(* IEC 61131-3 sources: Lasal/CPU_5344_V01/Class/Uitv_Regel_C, 1 file *)

(* ---- Uitv_Regel_C.st ---- *)
(*!
<Class
	Name               = "Uitv_Regel_C"
	Revision           = "0.0"
	RealtimeTask       = "false"
	CyclicTask         = "false"
	BackgroundTask     = "false"
	Sigmatek           = "false"
	OSInterface        = "false"
	HighPriority       = "false"
	Automatic          = "false"
	UpdateMode         = "Prescan"
	SharedCommandTable = "true"
	Objectsize         = "(330,840)">
	<Channels>
		<Server Name="actione" Visualized="true" Initialize="false" WriteProtected="true" Retentive="false"/>
		<Server Name="ClassSvr" Visualized="false" Initialize="false" WriteProtected="true" Retentive="false"/>
		<Server Name="ClassSvr0" Visualized="true" Initialize="false" WriteProtected="false" Retentive="false"/>
		<Server Name="Cmd" Visualized="true" Initialize="false" WriteProtected="true" Retentive="false"/>
		<Server Name="outputRule" Visualized="false" Initialize="true" WriteProtected="false" Retentive="false"/>
		<Server Name="Rnr" Visualized="true" Initialize="false" WriteProtected="true" Retentive="false"/>
		<Server Name="speed" Visualized="true" Initialize="false" WriteProtected="true" Retentive="false"/>
		<Server Name="UnitData" Visualized="true" Initialize="false" WriteProtected="true" Retentive="false"/>
		<Server Name="volgorde" Visualized="true" Initialize="false" WriteProtected="true" Retentive="false"/>
		<Server Name="x1pos" Visualized="true" Initialize="false" WriteProtected="true" Retentive="false"/>
		<Server Name="xy1Angle" Visualized="true" Initialize="false" WriteProtected="true" Retentive="false"/>
		<Server Name="xz1Angle" Visualized="true" Initialize="false" WriteProtected="true" Retentive="false"/>
		<Server Name="y1pos" Visualized="true" Initialize="false" WriteProtected="true" Retentive="false"/>
		<Server Name="z1pos" Visualized="true" Initialize="false" WriteProtected="true" Retentive="false"/>
		<Server Name="zy1Angle" Visualized="true" Initialize="false" WriteProtected="true" Retentive="false"/>
		<Client Name="list" Required="true" Internal="false"/>
		<Client Name="nextRegel" Required="false" Internal="false"/>
		<Client Name="RegelContent" Required="true" Internal="true"/>
		<Client Name="tMyBDintTODint1" Required="true" Internal="true"/>
	</Channels>
	<Network Name="Uitv_Regel_C">
		<!-- List of Components in this network -->
		<Components>
			<Object
				Name       = "RegelContent"
				Class      = "Uitv_Regel"
				Position   = "(420,150)"
				Visualized = "true">
				<Channels>
					<Server Name="actione"/>
					<Server Name="ClassSvr"/>
					<Server Name="Cmd"/>
					<Server Name="outputRule"/>
					<Server Name="Rnr"/>
					<Server Name="speed"/>
					<Server Name="Units"/>
					<Server Name="volgorde"/>
					<Server Name="x1pos"/>
					<Server Name="xy1Angle"/>
					<Server Name="xz1Angle"/>
					<Server Name="y1pos"/>
					<Server Name="z1pos"/>
					<Server Name="zy1Angle"/>
					<Client Name="list"/>
					<Client Name="nextRegel"/>
				</Channels>
			</Object>
			<Object
				Name       = "tMyBDintTODint1"
				Class      = "tMyBDintTODint"
				Position   = "(420,1140)"
				Visualized = "true">
				<Channels>
					<Server Name="ClassSvr"/>
					<Server Name="Data"/>
					<Client Name="cOutput"/>
				</Channels>
			</Object>
		</Components>
		<Comments>
		</Comments>
		<!-- List of Connections in this network -->
		<Connections>
			<Connection Source="this.RegelContent" Destination="RegelContent.ClassSvr"/>
			<Connection Source="RegelContent.nextRegel" Destination="this.nextRegel" Vertices="(420,240),(38,210),"/>
			<Connection Source="this.ClassSvr0" Destination="RegelContent.ClassSvr" Vertices="(908,270),(736,240),"/>
			<Connection Source="this.tMyBDintTODint1" Destination="tMyBDintTODint1.ClassSvr"/>
			<Connection Source="tMyBDintTODint1.cOutput" Destination="RegelContent.Units" Vertices="(420,1230),(330,1230),(330,1110),(840,1110),(840,420),(736,420),"/>
			<Connection Source="this.Rnr" Destination="RegelContent.Rnr" Vertices="(908,330),(736,300),"/>
			<Connection Source="this.Cmd" Destination="RegelContent.Cmd" Vertices="(908,390),(736,360),"/>
			<Connection Source="this.x1pos" Destination="RegelContent.x1pos" Vertices="(908,450),(736,480),"/>
			<Connection Source="this.y1pos" Destination="RegelContent.y1pos" Vertices="(908,510),(736,540),"/>
			<Connection Source="this.z1pos" Destination="RegelContent.z1pos" Vertices="(908,570),(736,600),"/>
			<Connection Source="this.zy1Angle" Destination="RegelContent.zy1Angle" Vertices="(908,630),(736,660),"/>
			<Connection Source="this.xz1Angle" Destination="RegelContent.xz1Angle" Vertices="(908,690),(736,720),"/>
			<Connection Source="this.xy1Angle" Destination="RegelContent.xy1Angle" Vertices="(908,750),(736,780),"/>
			<Connection Source="this.actione" Destination="RegelContent.actione" Vertices="(908,810),(736,840),"/>
			<Connection Source="this.speed" Destination="RegelContent.speed" Vertices="(908,870),(736,900),"/>
			<Connection Source="this.UnitData" Destination="tMyBDintTODint1.Data" Vertices="(908,930),(720,1290),"/>
			<Connection Source="this.volgorde" Destination="RegelContent.volgorde" Vertices="(908,990),(736,960),"/>
			<Connection Source="RegelContent.list" Destination="this.list" Vertices="(420,300),(38,270),"/>
			<Connection Source="this.outputRule" Destination="RegelContent.outputRule" Vertices="(908,1050),(736,1020),"/>
		</Connections>
		<!-- Headerfiles -->
		<Options>
		</Options>
	</Network>
</Class>
*)
Uitv_Regel_C : CLASS
  //Servers:
	ClassSvr 	: SvrChCmd_DINT;
	ClassSvr0 	: SvrCh_DINT;
	Rnr 	: SvrCh_DINT;
	Cmd 	: SvrCh_DINT;
	x1pos 	: SvrCh_DINT;
	y1pos 	: SvrCh_DINT;
	z1pos 	: SvrCh_DINT;
	zy1Angle 	: SvrCh_DINT;
	xz1Angle 	: SvrCh_DINT;
	xy1Angle 	: SvrCh_DINT;
	actione 	: SvrCh_DINT;
	speed 	: SvrCh_DINT;
	UnitData 	: SvrCh_tMyBDint;
	volgorde 	: SvrCh_DINT;
	outputRule 	: SvrCh_DINT;
  //Clients:
	nextRegel 	: CltCh_DINT;
	tMyBDintTODint1 	: CltChCmd_tMyBDintTODint;
	RegelContent 	: CltChCmd_Uitv_Regel;
	list 	: CltChCmd_GlobalList;
  //Variables:
  //Functions:

	FUNCTION VIRTUAL GLOBAL ClassSvr0::Read
		VAR_OUTPUT
			output (EAX) 	: DINT;
		END_VAR;

	FUNCTION VIRTUAL GLOBAL ClassSvr0::Write
		VAR_INPUT
			input (EAX) 	: DINT;
		END_VAR
		VAR_OUTPUT
			result (EAX) 	: DINT;
		END_VAR;

	FUNCTION VIRTUAL GLOBAL Rnr::Read
		VAR_OUTPUT
			output (EAX) 	: DINT;
		END_VAR;

	FUNCTION VIRTUAL GLOBAL Rnr::Write
		VAR_INPUT
			input (EAX) 	: DINT;
		END_VAR
		VAR_OUTPUT
			result (EAX) 	: DINT;
		END_VAR;

	FUNCTION VIRTUAL GLOBAL Cmd::Read
		VAR_OUTPUT
			output (EAX) 	: DINT;
		END_VAR;

	FUNCTION VIRTUAL GLOBAL Cmd::Write
		VAR_INPUT
			input (EAX) 	: DINT;
		END_VAR
		VAR_OUTPUT
			result (EAX) 	: DINT;
		END_VAR;

	FUNCTION VIRTUAL GLOBAL x1pos::Read
		VAR_OUTPUT
			output (EAX) 	: DINT;
		END_VAR;

	FUNCTION VIRTUAL GLOBAL x1pos::Write
		VAR_INPUT
			input (EAX) 	: DINT;
		END_VAR
		VAR_OUTPUT
			result (EAX) 	: DINT;
		END_VAR;

	FUNCTION VIRTUAL GLOBAL y1pos::Read
		VAR_OUTPUT
			output (EAX) 	: DINT;
		END_VAR;

	FUNCTION VIRTUAL GLOBAL y1pos::Write
		VAR_INPUT
			input (EAX) 	: DINT;
		END_VAR
		VAR_OUTPUT
			result (EAX) 	: DINT;
		END_VAR;

	FUNCTION VIRTUAL GLOBAL z1pos::Read
		VAR_OUTPUT
			output (EAX) 	: DINT;
		END_VAR;

	FUNCTION VIRTUAL GLOBAL z1pos::Write
		VAR_INPUT
			input (EAX) 	: DINT;
		END_VAR
		VAR_OUTPUT
			result (EAX) 	: DINT;
		END_VAR;

	FUNCTION VIRTUAL GLOBAL zy1Angle::Read
		VAR_OUTPUT
			output (EAX) 	: DINT;
		END_VAR;

	FUNCTION VIRTUAL GLOBAL zy1Angle::Write
		VAR_INPUT
			input (EAX) 	: DINT;
		END_VAR
		VAR_OUTPUT
			result (EAX) 	: DINT;
		END_VAR;

	FUNCTION VIRTUAL GLOBAL xz1Angle::Read
		VAR_OUTPUT
			output (EAX) 	: DINT;
		END_VAR;

	FUNCTION VIRTUAL GLOBAL xz1Angle::Write
		VAR_INPUT
			input (EAX) 	: DINT;
		END_VAR
		VAR_OUTPUT
			result (EAX) 	: DINT;
		END_VAR;

	FUNCTION VIRTUAL GLOBAL xy1Angle::Read
		VAR_OUTPUT
			output (EAX) 	: DINT;
		END_VAR;

	FUNCTION VIRTUAL GLOBAL xy1Angle::Write
		VAR_INPUT
			input (EAX) 	: DINT;
		END_VAR
		VAR_OUTPUT
			result (EAX) 	: DINT;
		END_VAR;

	FUNCTION VIRTUAL GLOBAL actione::Read
		VAR_OUTPUT
			output (EAX) 	: DINT;
		END_VAR;

	FUNCTION VIRTUAL GLOBAL actione::Write
		VAR_INPUT
			input (EAX) 	: DINT;
		END_VAR
		VAR_OUTPUT
			result (EAX) 	: DINT;
		END_VAR;

	FUNCTION VIRTUAL GLOBAL speed::Read
		VAR_OUTPUT
			output (EAX) 	: DINT;
		END_VAR;

	FUNCTION VIRTUAL GLOBAL speed::Write
		VAR_INPUT
			input (EAX) 	: DINT;
		END_VAR
		VAR_OUTPUT
			result (EAX) 	: DINT;
		END_VAR;

	FUNCTION VIRTUAL GLOBAL UnitData::Read
		VAR_OUTPUT
			output (EAX) 	: tMyBDint;
		END_VAR;

	FUNCTION VIRTUAL GLOBAL UnitData::Write
		VAR_INPUT
			input (EAX) 	: tMyBDint;
		END_VAR
		VAR_OUTPUT
			result (EAX) 	: tMyBDint;
		END_VAR;

	FUNCTION VIRTUAL GLOBAL volgorde::Read
		VAR_OUTPUT
			output (EAX) 	: DINT;
		END_VAR;

	FUNCTION VIRTUAL GLOBAL volgorde::Write
		VAR_INPUT
			input (EAX) 	: DINT;
		END_VAR
		VAR_OUTPUT
			result (EAX) 	: DINT;
		END_VAR;

	FUNCTION VIRTUAL GLOBAL outputRule::Read
		VAR_OUTPUT
			output (EAX) 	: DINT;
		END_VAR;

	FUNCTION VIRTUAL GLOBAL outputRule::Write
		VAR_INPUT
			input (EAX) 	: DINT;
		END_VAR
		VAR_OUTPUT
			result (EAX) 	: DINT;
		END_VAR;
  //Tables:
	FUNCTION @STD
		VAR_OUTPUT
			ret_code	: CONFSTATES;
		END_VAR;
	FUNCTION GLOBAL TAB @CT_;
END_CLASS;

#pragma using tMyBDintTODint
#pragma using Uitv_Regel
#pragma usingLtd GlobalList

FUNCTION VIRTUAL GLOBAL Uitv_Regel_C::ClassSvr0::Read
	VAR_OUTPUT
		output (EAX) 	: DINT;
	END_VAR

	ClassSvr0 := RegelContent.ClassSvr.Read();
	output := ClassSvr0;

END_FUNCTION

FUNCTION VIRTUAL GLOBAL Uitv_Regel_C::ClassSvr0::Write
	VAR_INPUT
		input (EAX) 	: DINT;
	END_VAR
	VAR_OUTPUT
		result (EAX) 	: DINT;
	END_VAR

	ClassSvr0 := input;
	result := (RegelContent.ClassSvr.Write(ClassSvr0))$DINT;

END_FUNCTION

FUNCTION VIRTUAL GLOBAL Uitv_Regel_C::Rnr::Read
	VAR_OUTPUT
		output (EAX) 	: DINT;
	END_VAR

	Rnr := RegelContent.Rnr.Read();
	output := Rnr;

END_FUNCTION

FUNCTION VIRTUAL GLOBAL Uitv_Regel_C::Rnr::Write
	VAR_INPUT
		input (EAX) 	: DINT;
	END_VAR
	VAR_OUTPUT
		result (EAX) 	: DINT;
	END_VAR

	Rnr := input;
	result := (RegelContent.Rnr.Write(Rnr))$DINT;

END_FUNCTION

FUNCTION VIRTUAL GLOBAL Uitv_Regel_C::Cmd::Read
	VAR_OUTPUT
		output (EAX) 	: DINT;
	END_VAR

	Cmd := RegelContent.Cmd.Read();
	output := Cmd;

END_FUNCTION

FUNCTION VIRTUAL GLOBAL Uitv_Regel_C::Cmd::Write
	VAR_INPUT
		input (EAX) 	: DINT;
	END_VAR
	VAR_OUTPUT
		result (EAX) 	: DINT;
	END_VAR

	Cmd := input;
	result := (RegelContent.Cmd.Write(Cmd))$DINT;

END_FUNCTION

FUNCTION VIRTUAL GLOBAL Uitv_Regel_C::x1pos::Read
	VAR_OUTPUT
		output (EAX) 	: DINT;
	END_VAR

	x1pos := RegelContent.x1pos.Read();
	output := x1pos;

END_FUNCTION

FUNCTION VIRTUAL GLOBAL Uitv_Regel_C::x1pos::Write
	VAR_INPUT
		input (EAX) 	: DINT;
	END_VAR
	VAR_OUTPUT
		result (EAX) 	: DINT;
	END_VAR

	x1pos := input;
	result := (RegelContent.x1pos.Write(x1pos))$DINT;

END_FUNCTION

FUNCTION VIRTUAL GLOBAL Uitv_Regel_C::y1pos::Read
	VAR_OUTPUT
		output (EAX) 	: DINT;
	END_VAR

	y1pos := RegelContent.y1pos.Read();
	output := y1pos;

END_FUNCTION

FUNCTION VIRTUAL GLOBAL Uitv_Regel_C::y1pos::Write
	VAR_INPUT
		input (EAX) 	: DINT;
	END_VAR
	VAR_OUTPUT
		result (EAX) 	: DINT;
	END_VAR

	y1pos := input;
	result := (RegelContent.y1pos.Write(y1pos))$DINT;

END_FUNCTION

FUNCTION VIRTUAL GLOBAL Uitv_Regel_C::z1pos::Read
	VAR_OUTPUT
		output (EAX) 	: DINT;
	END_VAR

	z1pos := RegelContent.z1pos.Read();
	output := z1pos;

END_FUNCTION

FUNCTION VIRTUAL GLOBAL Uitv_Regel_C::z1pos::Write
	VAR_INPUT
		input (EAX) 	: DINT;
	END_VAR
	VAR_OUTPUT
		result (EAX) 	: DINT;
	END_VAR

	z1pos := input;
	result := (RegelContent.z1pos.Write(z1pos))$DINT;

END_FUNCTION

FUNCTION VIRTUAL GLOBAL Uitv_Regel_C::zy1Angle::Read
	VAR_OUTPUT
		output (EAX) 	: DINT;
	END_VAR

	zy1Angle := RegelContent.zy1Angle.Read();
	output := zy1Angle;

END_FUNCTION

FUNCTION VIRTUAL GLOBAL Uitv_Regel_C::zy1Angle::Write
	VAR_INPUT
		input (EAX) 	: DINT;
	END_VAR
	VAR_OUTPUT
		result (EAX) 	: DINT;
	END_VAR

	zy1Angle := input;
	result := (RegelContent.zy1Angle.Write(zy1Angle))$DINT;

END_FUNCTION

FUNCTION VIRTUAL GLOBAL Uitv_Regel_C::xz1Angle::Read
	VAR_OUTPUT
		output (EAX) 	: DINT;
	END_VAR

	xz1Angle := RegelContent.xz1Angle.Read();
	output := xz1Angle;

END_FUNCTION

FUNCTION VIRTUAL GLOBAL Uitv_Regel_C::xz1Angle::Write
	VAR_INPUT
		input (EAX) 	: DINT;
	END_VAR
	VAR_OUTPUT
		result (EAX) 	: DINT;
	END_VAR

	xz1Angle := input;
	result := (RegelContent.xz1Angle.Write(xz1Angle))$DINT;

END_FUNCTION

FUNCTION VIRTUAL GLOBAL Uitv_Regel_C::xy1Angle::Read
	VAR_OUTPUT
		output (EAX) 	: DINT;
	END_VAR

	xy1Angle := RegelContent.xy1Angle.Read();
	output := xy1Angle;

END_FUNCTION

FUNCTION VIRTUAL GLOBAL Uitv_Regel_C::xy1Angle::Write
	VAR_INPUT
		input (EAX) 	: DINT;
	END_VAR
	VAR_OUTPUT
		result (EAX) 	: DINT;
	END_VAR

	xy1Angle := input;
	result := (RegelContent.xy1Angle.Write(xy1Angle))$DINT;

END_FUNCTION

FUNCTION VIRTUAL GLOBAL Uitv_Regel_C::actione::Read
	VAR_OUTPUT
		output (EAX) 	: DINT;
	END_VAR

	actione := RegelContent.actione.Read();
	output := actione;

END_FUNCTION

FUNCTION VIRTUAL GLOBAL Uitv_Regel_C::actione::Write
	VAR_INPUT
		input (EAX) 	: DINT;
	END_VAR
	VAR_OUTPUT
		result (EAX) 	: DINT;
	END_VAR

	actione := input;
	result := (RegelContent.actione.Write(actione))$DINT;

END_FUNCTION

FUNCTION VIRTUAL GLOBAL Uitv_Regel_C::speed::Read
	VAR_OUTPUT
		output (EAX) 	: DINT;
	END_VAR

	speed := RegelContent.speed.Read();
	output := speed;

END_FUNCTION

FUNCTION VIRTUAL GLOBAL Uitv_Regel_C::speed::Write
	VAR_INPUT
		input (EAX) 	: DINT;
	END_VAR
	VAR_OUTPUT
		result (EAX) 	: DINT;
	END_VAR

	speed := input;
	result := (RegelContent.speed.Write(speed))$DINT;

END_FUNCTION

FUNCTION VIRTUAL GLOBAL Uitv_Regel_C::UnitData::Read
	VAR_OUTPUT
		output (EAX) 	: tMyBDint;
	END_VAR

	UnitData := tMyBDintTODint1.Data.Read();
	output := UnitData;

END_FUNCTION

FUNCTION VIRTUAL GLOBAL Uitv_Regel_C::UnitData::Write
	VAR_INPUT
		input (EAX) 	: tMyBDint;
	END_VAR
	VAR_OUTPUT
		result (EAX) 	: tMyBDint;
	END_VAR

	UnitData := input;
	result := (tMyBDintTODint1.Data.Write(UnitData))$tMyBDint;

END_FUNCTION

FUNCTION VIRTUAL GLOBAL Uitv_Regel_C::volgorde::Read
	VAR_OUTPUT
		output (EAX) 	: DINT;
	END_VAR

	volgorde := RegelContent.volgorde.Read();
	output := volgorde;

END_FUNCTION

FUNCTION VIRTUAL GLOBAL Uitv_Regel_C::volgorde::Write
	VAR_INPUT
		input (EAX) 	: DINT;
	END_VAR
	VAR_OUTPUT
		result (EAX) 	: DINT;
	END_VAR

	volgorde := input;
	result := (RegelContent.volgorde.Write(volgorde))$DINT;

END_FUNCTION

FUNCTION VIRTUAL GLOBAL Uitv_Regel_C::outputRule::Read
	VAR_OUTPUT
		output (EAX) 	: DINT;
	END_VAR

	outputRule := RegelContent.outputRule.Read();
	output := outputRule;

END_FUNCTION

FUNCTION VIRTUAL GLOBAL Uitv_Regel_C::outputRule::Write
	VAR_INPUT
		input (EAX) 	: DINT;
	END_VAR
	VAR_OUTPUT
		result (EAX) 	: DINT;
	END_VAR

	outputRule := input;
	result := (RegelContent.outputRule.Write(outputRule))$DINT;

END_FUNCTION
